// TIA Portal V19 export
VAR_GLOBAL   // PLC tag table "Default tag table"
   Tag_1 AT %M100.0 : Bool;
   Tag_2 AT %M100.1 : Bool;
END_VAR
